(*
Nazwa:		FB_FormsDragStepper
Opis:		Przeciąganie formatek 
Wersja:		V0.22
Data:		2025-09-04
Autor:		DJ, DP
Urządzenia:	Siłownik podnoszenia wideł, Silnik krokowy przeciągania 
Ostatnie zmiany:
	- 20250904 [DP] EventLog->wywołać błędy 
	- 2025-08-19 [DP] Homing false
	- 2024-11-25 [DP] Czujnik dół
	- 2024-10-01 [DP] ESTOP Delay
	- RRRR-MM-DD [KTO?] Tekst Tekst Tekst Tekst Tekst Tekst Tekst Tekst Tekst Tekst 
	- 2025-09-15[VS] Jazda i stop w pozycji końcowej
Konfiguracja:
	- Krokówka
	Instukcja:
		-
		-
		-
	
Info:
	- Obsługa tylko jednego siłownika podnoszenia i dwóch siłowników prowadzących

*)

FUNCTION_BLOCK FB_FormsDragStepper
VAR_INPUT
	bEnable										: BOOL;				//Zezwolenie na pracę
	bEStop										: BOOL;				//Stop awaryjny włączony
	bRun										: BOOL;				//Rozkaz przeciagania
	bPrepare									: BOOL;				//Rozkaz przygotownaia 
	bDragUpWhenReady							: BOOL;					
	bHoming										: BOOL;				//Zezwolenie na wykonanie bazowania i pozycjonowanie układu
	bHomingDirection							: BOOL;				//Kierunek bazowania
	bBefore2ActuatorOff							: BOOL;
	bDelayAfterDrag								: BOOL;				//Opóżnienie po przeciąganiu
	bHeightSet									: BOOL;				//Ustaw do pozycji
	bIgnoreError								: BOOL;				//Ignorowanie błędów 
	bReset										: BOOL;				//Reset błędu, jeśli jest w stanie "eError"
	bResetCycle									: BOOL;				//Reset cyklu

	bTwoPhaseMode								: BOOL;				//Załączone dozowanie dwufazowe
	lrMinPosition								: LREAL;			 	
	lrMaxPosition								: LREAL;			 		
	lrStartPosition								: LREAL;			//Zadane położenie 
	lrMiddlePosition							: LREAL;			//Zadane położenie 
	lrEndPosition								: LREAL;			//Zadane położenie 		
	lrStartPositionTwoPhase						: LREAL;			//Zadane położenie 
	lrMiddlePositionTwoPhase					: LREAL;			//Zadane położenie 
	lrEndPositionTwoPhase						: LREAL;			//Zadane położenie 	
	lrLeadActuatorMoveUpPosition				: LREAL;			//Zadane położenie 	
	lrDragAcceleration							: LREAL;			//Przyspieszenie 
	lrDragDeceleration							: LREAL;			//Opóźnienie 
	lrDragJerk									: LREAL;			//Jerk
	lrDragSpeed									: LREAL;			//Prędkość 
	
	bHomingSensor								: BOOL;				//Czujnik bazowania 
	bDragUpSensor								: BOOL;				//
	bDragDownSensor								: BOOL;				//
	bLead1UpSensor								: BOOL;				//
	bLead2UpSensor								: BOOL;				//
	bManualMovement								: BOOL;				//Zezwolenie na ruchy ręczne

	_ALARMINFO_									: BOOL;
	iStationIndex								: UDINT;
	wsStationName								: WSTRING;
	bMoveToEndPosition							: BOOL;					//ustawienie w końcowej pozycji dla uruchomienia
END_VAR

VAR_OUTPUT
	eState										: E_Station;
	eRunningState								: E_DragStationState;	// Stan przeciągania formatek
	bError										: BOOL;					// Błąd stacji
	udiErrorID									: UDINT;				// Nr blędu przeciągania formatek
	sErrorDescription							: STRING(200);			// Opis błędu
	sErrorDescription2							: STRING(200);			// Opis błędu
	sErrorStationName							: STRING;				// Nazwa stacji
	udiStationID								: UDINT;				// Nr stacji

	bDragActuator								: BOOL;					
	bLeadBefore1Actuator						: BOOL;					
	bLeadBefore2Actuator						: BOOL;					
	
	bCycleDone									: BOOL;					//Sygnał zakończenia cyklu
	bCycleNotDone								: BOOL;
	bHomingDone									: BOOL;
	tCycleTime									: TIME;					//Czas cyklu
	lrActualDragPosition						: LREAL;				//Aktualne położenie
	//Dodatkowe	
	eRunningStateBeforeEStop					: E_DragStationState;	//Stan przed E-Stopem	
	bWasErrorOrEstop							: BOOL;
	
END_VAR

VAR
	(*LastStates*)
	eLastState									: E_Station;						//Stan ogólny bloku
	eLastStateTemp								: E_Station;						//Stan ogólny bloku
	eLastRunningState							: E_DragStationState;				//Stan podbloku
	eLastRunningStateTemp						: E_DragStationState;				//Stan podbloku
	
	(*Axis online*)
	fbDrag										: FB_McAxisOnlineNC;
	stDrag										: ST_McAxisOnline;
	                                    		                                 		
	(*Control*)
	tonResetting								: TON;								//Czas resetu
	tonHoming									: TON;
	tonPreparingToReady							: TON;								//Czas potrzeby na przygotowanie osi
	rtResetCommands								: R_TRIG;                                    	
	rtResetCycle								: R_TRIG;

	(*Statistics*)
	tonCycleTimer								: TON;								//Czas cyklu przeciągania	
	rtrigCycleTimerRead							: R_TRIG;

	(*Homing*)
	iHomingCase									: INT;
	
	(*Aborting*)
	iAbortingCase								: INT;
	                                    	
	(*Errors*)
	bStateError									: BOOL;
	tonEstopDelay								: TON;
	bResetCycleOn								: BOOL;
	tonbDragUpSensor							: TON;	
	tonbDragDownSensor							: TON;		
	tonbLead1UpSensor							: TON;
	tonbLead2UpSensor							: TON;
	
	(*Running*)

	tonNotDragActuatorDelay						: TON;
	tonRunningDraging							: TON;
	tonRunningeEndingOfDrag						: TON;
	(*Inne*)
	
		//Zmienne od EVENTLOGGER
	bAlarmInit 						: BOOL := TRUE; 
	nAlarmNumerator					: INT;
	arfbAlarm						: ARRAY[0..19] OF  FB_TcAlarm;		//Tablica bloczków błędów
	fbSourceInfo 					: FB_TcSourceInfo;
	iSourceInfo						: I_TcSourceInfo;
	sAlarmTest						: STRING;
	//Koniec zmiennych od EVENTLOGGER
	
END_VAR
	
VAR_IN_OUT
	bManualDragActuator							: BOOL;		
	bManualLeadBefore1Actuator					: BOOL;			
	bManualLeadBefore2Actuator					: BOOL;			
	bManualDragRight							: BOOL;				
	bManualDragLeft								: BOOL;		
	DragAxisRef									: AXIS_REF;		
END_VAR

ResetAll();
ErrorHandling();
Signals();
Control();
Limits();
DragControlBlocks();
Statistics();
aStationID();
(*Zapisywanie ostatniego stanu*)
IF eLastStateTemp<>eState THEN
	eLastState := eLastStateTemp;
END_IF
eLastStateTemp := eState;
IF eLastRunningStateTemp<>eRunningState THEN
	eLastRunningState := eLastRunningStateTemp;
END_IF
eLastRunningStateTemp := eRunningState;
(*Koniec Zapisywanie ostatniego stanu*)

ACTION aStationID:
udiStationID	:=	iStationIndex;
END_ACTION

ACTION Control:


	(*****Wyłączenie enable*****)
	IF NOT bEnable AND NOT bError THEN
		IF eState <> E_Station.eDisabled AND eState <> E_Station.ePreparingToDisable THEN
				eState 								:= E_Station.ePreparingToDisable; 
		END_IF	
	END_IF

	(*****Estop*****)
	IF NOT bEstop  THEN	
		IF eState <> E_Station.eAborted AND eState <> E_Station.eAborting AND eState <> E_Station.eDisabled THEN
				eRunningStateBeforeEStop			:= eRunningState;
				eState 								:= E_Station.eAborting; 
				iAbortingCase						:= 0; 
		END_IF
	END_IF


	
CASE eState OF
	
//==========================================================================================	
	E_Station.eDisabled: 						// Stan nieaktywnosci (Stacja wyłączona) 
		
		IF bEnable THEN
			eState 									:= E_Station.ePreparingToReady; 
		END_IF 

//==========================================================================================	    
	E_Station.eAborted: 						// Stan bezpiecznego zatrzymania (po Abortingu) 	
			
		IF bEStop THEN
			bWasErrorOrEstop						:= TRUE;	
			eState 									:= E_Station.ePreparingToReady;
		END_IF		
			
//==========================================================================================	
	E_Station.eAborting:                 		// Stan bezpiecznego zatrzymywania (po EStopie)
		
		CASE iAbortingCase OF
			
			0: //Inicjalizacja
				IF stDrag.mcPower.bStatus THEN
					iAbortingCase					:= 10;
				ELSE
					iAbortingCase					:= 40;
				END_IF
				
			10: //Komenda MC_STOP
				stDrag.mcStop.bExecute				:= TRUE;	
				//Czekam na Done
				IF stDrag.mcStop.bDone THEN
					stDrag.mcStop.bExecute			:= FALSE;
					iAbortingCase					:= 20;
				END_IF
				
			20: //Kasowanie komend
				stDrag.mcMoveAbsolute.bExecute		:= FALSE;
				stDrag.mcMoveRelative.bExecute		:= FALSE;
				ResetCommands();
				iAbortingCase						:= 30;
	
			30: //Wyłączenie osi
				stDrag.mcPower.bEnable				:= FALSE;
				stDrag.mcPower.bEnable_Negative		:= FALSE;
				stDrag.mcPower.bEnable_Positive		:= FALSE;
				IF NOT stDrag.mcPower.bStatus THEN
					iAbortingCase					:= 40;
				END_IF
				
			40: //Kasowanie podzespołow
				ResetCommands();
				iAbortingCase						:= 50;
				
			50: //Przejście do Aborted
				iAbortingCase						:= 0;
				eState								:= E_Station.eAborted;
				eRunningState						:= E_DragStationState.eReady;
				
		END_CASE

//==========================================================================================			
	E_Station.eError:                 	 		// Stan błędu 	
		
		bWasErrorOrEstop							:= TRUE;

		IF bReset THEN
			eState									:= E_Station.eResetting;	
		ELSE
			ResetCommands();
		END_IF
			
//==========================================================================================
	E_Station.eResetting:						// Stan resetowania bledu (po Errorze)
			
	//Procedura obsługi resetu w zależności od błędu
//	CASE udiErrorID OF 
//	CASE udiErrorID - iStationIndex(*udiResetStep*) OF 	
//		171: //Error 1 - Błąd Serwa
		IF  arfbAlarm[0].bActive THEN
			stDrag.mcReset.bExecute					:= TRUE;
			IF stDrag.mcReset.bDone THEN
				stDrag.mcReset.bExecute				:= FALSE;
				bError								:= FALSE;
			END_IF	
		END_IF
		
//		172,173://Error 2 - Błąd siłownika przeciągania
		IF  arfbAlarm[1].bActive OR arfbAlarm[2].bActive THEN
			bDragActuator							:= FALSE;	
			//bLeadBefore1Actuator					:= FALSE;				
			//bLeadBefore2Actuator					:= FALSE;			
			bError									:= FALSE;
		END_IF	
// 		174: //Error 4 - Błąd siłownika prowadzenia
		IF arfbAlarm[3].bActive THEN
			//bDragActuator							:= FALSE;	
			bLeadBefore1Actuator					:= TRUE;				
			//bLeadBefore2Actuator					:= FALSE;			
			bError									:= FALSE;		
		END_IF
// 		175: //Error 5 - Błąd siłownika prowadzenia
		IF arfbAlarm[4].bActive THEN
			//bDragActuator							:= FALSE;	
			bLeadBefore2Actuator					:= NOT bBefore2ActuatorOff;				
			//bLeadBefore2Actuator					:= FALSE;			
			bError									:= FALSE;		
		END_IF
//	END_CASE
	
	IF NOT bError THEN
		udiErrorID									:= 0;
		sErrorDescription							:= '';
		sErrorDescription2							:= '';	
		eState										:= E_Station.ePreparingToReady;
	ELSIF tonResetting.Q THEN                   	
		eState										:= E_Station.eError;
	END_IF	
 
//==========================================================================================
	E_Station.eManualMovement:     				// Stan ruchów manualnych  
       
		ManualMovements();
		//Wyjście z trybu serwisowego
		IF NOT bManualMovement THEN
			bDragActuator							:=	bManualDragActuator;	
			bLeadBefore1Actuator					:=	bManualLeadBefore1Actuator;
			bLeadBefore2Actuator					:=	bManualLeadBefore2Actuator;
			eState									:=	E_Station.eReady;
		END_IF 

//==========================================================================================		
	E_Station.eHoming:							// Stan bazowania 
		
		Homing();	
		IF NOT bHoming AND NOT bHeightSet AND tonHoming.Q THEN
			eState									:=	E_Station.ePreparingToReady;
		END_IF		
			
//==========================================================================================
	E_Station.eHomingDone:                  	// Stan wykonania bazowania 

		bHomingDone									:= TRUE;
		bResetCycleOn								:= FALSE;		
		IF NOT bHoming AND NOT bHeightSet AND NOT bResetCycleOn THEN
		//	eState									:=	E_Station.eReady;
			eState									:=	E_Station.ePreparingToReady;
		END_IF

//==========================================================================================
	E_Station.ePreparingToReady:            	// Stan przygotowywania do gotowosci (zawsze przed Ready)  

		IF tonPreparingToReady.Q THEN
			
			stDrag.mcPower.bEnable					:= TRUE;
			stDrag.mcPower.bEnable_Negative			:= TRUE;
			stDrag.mcPower.bEnable_Positive			:= TRUE;
			stDrag.mcPower.lrOverride				:= 100;
			
			IF stDrag.mcPower.bStatus THEN
				
				ResetCommands();
				eState								:= E_Station.eReady;
				eRunningState						:= E_DragStationState.eReady;
				
				IF bResetCycleOn THEN
					eState							:= E_Station.eHoming;
				END_IF
				
			END_IF
		
		END_IF			

//==========================================================================================
	E_Station.ePreparingToDisable:         	 	// Stan przygotowywania do nieaktywnosci (po wyłączeniu Enable) 
  
		stDrag.mcPower.bEnable						:= FALSE;
		stDrag.mcPower.bEnable_Negative				:= FALSE;
		stDrag.mcPower.bEnable_Positive				:= FALSE;
		stDrag.mcPower.lrOverride					:= 0;
		
		bWasErrorOrEstop							:= FALSE;
		bHomingDone									:= FALSE;	
		
		IF NOT stDrag.mcPower.bStatus THEN
			ResetCommands();
			eState									:= 	E_Station.eDisabled;
			eRunningState							:= 	E_DragStationState.eReady;
		END_IF

//==========================================================================================	
	E_Station.eReady:							// Stan gotowosci 


		(*Skasowanie wszystkich komend*)
		IF rtResetCommands.Q THEN	ResetCommands();	END_IF		
		
		IF bDragUpWhenReady THEN
			bDragActuator							:=	TRUE;
		END_IF
	
		IF (bRun OR bPrepare) AND NOT bCycleDone THEN
			eState									:= E_Station.eStarting;
			//IF bDragUpWhenReady THEN
				bDragActuator						:=	FALSE;
			//END_IF			
		END_IF		
		IF bHoming OR bHeightSet THEN
			eState									:= E_Station.eHoming;
		END_IF
		IF bManualMovement THEN
			bManualDragActuator						:=	bDragActuator;			
			bManualLeadBefore1Actuator				:=	bLeadBefore1Actuator;	
			bManualLeadBefore2Actuator				:=	bLeadBefore2Actuator;	
			bManualDragRight						:=	FALSE;		
			bManualDragLeft							:=	FALSE;					
			eState									:= E_Station.eManualMovement;					
		END_IF
		IF NOT bRun AND NOT bPrepare THEN
			bCycleDone								:= FALSE;
		END_IF

//==========================================================================================
	E_Station.eStopping:					// Stan zatrzymywania 
		
		Running();
		
		//Czekam dopóki skończy ruch
		IF	eRunningState <> E_DragStationState.eDraging AND eRunningState <> E_DragStationState.eDragingDone AND eRunningState <> E_DragStationState.eEndingOfDrag AND eRunningState <> E_DragStationState.eDraged
		AND  eRunningState <> E_DragStationState.eEndingOfDragDone AND  eRunningState <> E_DragStationState.eLowering  THEN	
			stDrag.mcReset.bExecute					:= TRUE;	
		END_IF
		
		//Reset ruchu
		IF stDrag.mcReset.bDone THEN		
			stDrag.mcReset.bExecute					:= FALSE;
			eState 									:= E_Station.eReady;
		END_IF

//==========================================================================================
	E_Station.eStarting:                  	// Stan uruchamiania (po Ready)
		
		eState										:= E_Station.eRunning;

//==========================================================================================
	E_Station.eRunning:               		// Stan wykonywania cyklu (po Startingu), w tym stanie osobny
 
		Running();

		IF NOT bRun AND NOT bPrepare THEN					(*Przerywanie cyklu*)
			eState 				 					:= E_Station.eStopping;	
		END_IF
			
		IF bCycleDone THEN (*Cykl zakończony*)
			eState 				 					:= E_Station.eReady;
		END_IF	
		
//==========================================================================================
END_CASE
END_ACTION

ACTION DragControlBlocks:
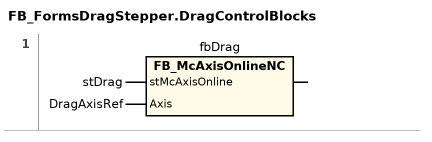
// NETWORK 1
fbDrag(stMcAxisOnline := stDrag, Axis := DragAxisRef); // FB_McAxisOnlineNC
END_ACTION

ACTION ErrorHandling:
// Alarm_0260	260	Error	Błąd napędu przeciągania. Błąd NC: {0}
// Alarm_0261	261	Error	Siłownik przeciągania | Blokada podnoszenia - sprawdź czujnik lub odblokuj
// Alarm_0262	262	Error	Siłownik przeciągania | Blokada opuszczania siłownika - sprawdź czujnik lub odblokuj
// Alarm_0263	263	Error	Siłownik prowadzenia | Blokada podnoszenia - sprawdź czujnik lub odblokuj
// Alarm_0264	264	Error	Siłownik prowadzenia | Blokada podnoszenia - sprawdź czujnik lub odblokuj

IF bAlarmInit THEN
    bAlarmInit := FALSE; 
	fbSourceInfo.Clear();
	fbSourceInfo.sName:=wsLiteral_TO_UTF8(wsStationName);//'Machine';
	fbSourceInfo.nId:=iStationIndex;//2700;
	// Alarm_0260	260	Error	Błąd napędu przeciągania. Błąd NC: {0}
    arfbAlarm[0].CreateEx(stEventEntry := TC_EVENTS.AlarmClass.Alarm_0260, bWithConfirmation:= FALSE,  ipSourceInfo:= fbSourceInfo); 
	// Alarm_0261	261	Error	Siłownik przeciągania | Blokada podnoszenia - sprawdź czujnik lub odblokuj
	arfbAlarm[1].CreateEx(stEventEntry := TC_EVENTS.AlarmClass.Alarm_0261, bWithConfirmation:= FALSE,  ipSourceInfo:= fbSourceInfo);
	// Alarm_0262	262	Error	Siłownik przeciągania | Blokada opuszczania siłownika - sprawdź czujnik lub odblokuj
	arfbAlarm[2].CreateEx(stEventEntry := TC_EVENTS.AlarmClass.Alarm_0262, bWithConfirmation:= FALSE,  ipSourceInfo:= fbSourceInfo);
	// Alarm_0263	263	Error	Siłownik prowadzenia | Blokada podnoszenia - sprawdź czujnik lub odblokuj
	arfbAlarm[3].CreateEx(stEventEntry := TC_EVENTS.AlarmClass.Alarm_0263, bWithConfirmation:= FALSE,  ipSourceInfo:= fbSourceInfo);
	// Alarm_0264	264	Error	Siłownik prowadzenia | Blokada podnoszenia - sprawdź czujnik lub odblokuj
	arfbAlarm[4].CreateEx(stEventEntry := TC_EVENTS.AlarmClass.Alarm_0264, bWithConfirmation:= FALSE,  ipSourceInfo:= fbSourceInfo);

	
END_IF

//CZYTANIE STATUSÓW
DragAxisRef.ReadStatus();

bStateError										:= (eState=E_Station.eError) OR (eState=E_Station.eResetting) OR NOT bEstop OR bIgnoreError;
tonEstopDelay									(IN:=bEStop,	PT:=T#4S);

IF bEnable AND tonEstopDelay.Q THEN
	// Alarm_0260	260	Error	Błąd napędu przeciągania. Błąd NC: {0}
	//Error 1 - Błąd Serwa
	IF stDrag.bError THEN
		bHomingDone									:= FALSE;	
		arfbAlarm[0].ipArguments.Clear() .AddString(stDrag.stError.sNcError);
		IF NOT arfbAlarm[0].bActive THEN
			stDrag.mcReset.bExecute				:= TRUE; // na testy jak wystąpi błąd
			arfbAlarm[0].Raise(nTimeStamp:=0);
		END_IF
	ELSE	
		IF  arfbAlarm[0].bActive AND bReset THEN
			arfbAlarm[0].Clear(nTimeStamp:=0, bResetConfirmation:= FALSE);
		END_IF	
// 		stDrag.mcReset.bExecute				:= TRUE; // na testy jak wystąpi błąd
// 		bError								:= TRUE;
// 		udiErrorID							:= 171;
// 		//udiErrorID							:= udiErrorID + iStationIndex;
// 		sErrorDescription					:= 'Błąd napędu przeciągania. Błąd NC:';
// 		sErrorDescription2					:= stDrag.stError.sNcError;
	END_IF
	
	//Alarm_0261	261	Error	Siłownik przeciągania | Blokada podnoszenia - sprawdź czujnik lub odblokuj
	//Error 2 - Błąd siłownika przeciągania
	tonbDragUpSensor	(IN:= bDragActuator AND NOT bDragUpSensor	, PT:=T#2S);
	IF tonbDragUpSensor.Q THEN
		bHomingDone									:= FALSE;			
		IF NOT arfbAlarm[1].bActive THEN
			arfbAlarm[1].Raise(nTimeStamp:=0);
		END_IF
	ELSE	
		IF  arfbAlarm[1].bActive AND bReset THEN
			arfbAlarm[1].Clear(nTimeStamp:=0, bResetConfirmation:= FALSE);
		END_IF	
// 		bError								:= TRUE;
// 		udiErrorID							:= 172;	
// 		//udiErrorID 							:= udiErrorID + iStationIndex;
// 		sErrorDescription					:= 'Siłownik przeciągania';
// 		sErrorDescription2					:= 'Blokada podnoszenia - sprawdź czujnik lub odblokuj';
	END_IF
	
	// Alarm_0262	262	Error	Siłownik przeciągania | Blokada opuszczania siłownika - sprawdź czujnik lub odblokuj
	//Error 3 - Błąd siłownika przeciągania
	tonbDragDownSensor	(IN:= NOT bDragActuator AND NOT bDragDownSensor	AND bRun, PT:=T#2S);
	IF tonbDragDownSensor.Q THEN
		IF NOT arfbAlarm[2].bActive THEN
			arfbAlarm[2].Raise(nTimeStamp:=0);
		END_IF
	ELSE	
		IF  arfbAlarm[2].bActive AND bReset THEN
			arfbAlarm[2].Clear(nTimeStamp:=0, bResetConfirmation:= FALSE);
		END_IF	
// 		bError								:= TRUE;
// 		udiErrorID							:= 173;	
// 		//udiErrorID 							:= udiErrorID + iStationIndex;
// 		sErrorDescription					:= 'Siłownik przeciągania';
// 		sErrorDescription2					:= 'Blokada opuszczania siłownika - sprawdź czujnik lub odblokuj';
	END_IF;			
	
	// Alarm_0263	263	Error	Siłownik prowadzenia | Blokada podnoszenia - sprawdź czujnik lub odblokuj
	//Error 4 - Błąd siłownika prowadzenia
	tonbLead1UpSensor	(IN:= bLeadBefore1Actuator AND NOT bLead1UpSensor	, PT:=T#2S);
	IF tonbLead1UpSensor.Q THEN
		IF NOT arfbAlarm[3].bActive THEN
			arfbAlarm[3].Raise(nTimeStamp:=0);
		END_IF
	ELSE	
		IF  arfbAlarm[3].bActive AND bReset THEN
			arfbAlarm[3].Clear(nTimeStamp:=0, bResetConfirmation:= FALSE);
		END_IF	
// 		bError								:= TRUE;
// 		udiErrorID							:= 174;	
// 		//udiErrorID 							:= udiErrorID + iStationIndex;
// 		sErrorDescription					:= 'Siłownik prowadzenia';
// 		sErrorDescription2					:= 'Blokada podnoszenia - sprawdź czujnik lub odblokuj';
	END_IF;		
	
	//// Alarm_0264	264	Error	Siłownik prowadzenia | Blokada podnoszenia - sprawdź czujnik lub odblokuj
	//Error 5 - Błąd siłownika prowadzenia
	tonbLead2UpSensor	(IN:= bLeadBefore2Actuator AND NOT bLead2UpSensor	, PT:=T#2S);
	IF tonbLead2UpSensor.Q THEN
		IF NOT arfbAlarm[4].bActive THEN
			arfbAlarm[4].Raise(nTimeStamp:=0);
		END_IF
	ELSE	
		IF  arfbAlarm[4].bActive AND bReset THEN
			arfbAlarm[4].Clear(nTimeStamp:=0, bResetConfirmation:= FALSE);
		END_IF	
// 		bError								:= TRUE;
// 		udiErrorID							:= 175;	
// 		//udiErrorID 							:= udiErrorID + iStationIndex;
// 		sErrorDescription					:= 'Siłownik prowadzenia';
// 		sErrorDescription2					:= 'Blokada podnoszenia - sprawdź czujnik lub odblokuj';
	END_IF;		
ELSE
	bError := FALSE;
END_IF

//******************PRZEJŚCIE DO eERROR*****************************

IF bError AND  NOT bStateError THEN
	eState 									:= E_Station.eError;
END_IF

//****************WYŚWIETLANIE STATUSU BLEDU************************
(*Wyświetlanie błedu na wyjściu*)
bError							:= FALSE;
FOR nAlarmNumerator := 0 TO 19 DO
	bError						:= bError OR arfbAlarm[nAlarmNumerator].bActive;
END_FOR

(*Przepisywanie nazwy stacji*)
sErrorStationName 							:= WSTRING_TO_STRING(wsStationName);
END_ACTION

ACTION Homing:

stDrag.mcMoveRelative.lrAcceleration			:=	1500;
stDrag.mcMoveRelative.lrDeceleration			:=	1500;
stDrag.mcMoveRelative.lrJerk					:=	15000;
stDrag.mcMoveRelative.lrVelocity				:=	15;

stDrag.mcMoveVelocity.lrAcceleration			:= 	2500;
stDrag.mcMoveVelocity.lrDeceleration			:= 	2500;
stDrag.mcMoveVelocity.lrJerk					:= 	2500;
stDrag.mcMoveVelocity.lrVelocity				:= 	10;	

stDrag.stStatus.lrPosDiff;
stdrag.stStatus.lrActPos;

IF bHoming THEN // Bazowanie - podjazd do góry i ustawienie obrotu
	CASE iHomingCase OF
	
	0: //Opuszczamy widły
		bHomingDone										:= FALSE;
		                                        		
		stDrag.mcMoveAbsolute.bExecute					:= FALSE;
		stDrag.mcMoveRelative.bExecute					:= FALSE;
		stDrag.mcMoveVelocity.bExecute					:= FALSE;
		
		bDragActuator									:= FALSE;	
		bLeadBefore1Actuator							:= TRUE; 	
		bLeadBefore2Actuator							:= NOT bBefore2ActuatorOff;
			
		iHomingCase										:= 10;
	
	10: //Sprawdzamy czy jest na czujniku
		IF bHomingSensor THEN
			iHomingCase									:= 20;
		ELSE                                        	
			iHomingCase									:= 30;
		END_IF
		
	20: //Muszę wyjechać z czujnika
		stDrag.mcMoveRelative.lrAcceleration			:=1500;
		stDrag.mcMoveRelative.lrDeceleration			:=1500;
		stDrag.mcMoveRelative.lrJerk					:=15000;
		stDrag.mcMoveRelative.lrVelocity				:=15;

		stDrag.mcMoveRelative.lrDistance				:= 50; // bylo 50
		IF bHomingDirection THEN
			stDrag.mcMoveRelative.lrDistance			:= -50; // bylo 50
		END_IF
		
		stDrag.mcMoveRelative.bExecute					:= TRUE;
		
		IF stDrag.mcMoveRelative.bDone THEN
			stDrag.mcMoveRelative.bExecute				:= FALSE;
			iHomingCase									:= 30;
		END_IF
		
	30: //Bazuje na czujnik
		stDrag.mcMoveVelocity.lrAcceleration			:= 2500;
		stDrag.mcMoveVelocity.lrDeceleration			:= 2500;
		stDrag.mcMoveVelocity.lrJerk					:= 2500;
		stDrag.mcMoveVelocity.lrVelocity				:= 10;	
	
		stDrag.mcMoveVelocity.eDirection				:= MC_Negative_Direction;
		IF bHomingDirection THEN
			stDrag.mcMoveVelocity.eDirection			:= MC_Positive_Direction;
		END_IF
		
		stDrag.mcMoveVelocity.bExecute					:= TRUE;
		
		IF bHomingSensor THEN
			stDrag.mcMoveVelocity.bExecute				:= FALSE;
			iHomingCase									:= 40;
		END_IF
		
	40: //Zatrzymanie osi
		stDrag.mcStop.bExecute							:= TRUE;
		
		IF stDrag.mcStop.bDone THEN
			stDrag.mcStop.bExecute						:= FALSE;
			iHomingCase									:= 50;
		END_IF
	
	50: 

		iHomingCase										:= 60;
		
	60: //Bazujemy Enkoder
		stDrag.mcHome.eHomingMode						:= MC_Direct;
		stDrag.mcHome.lrPosition						:= lrMinPosition;
		IF bHomingDirection THEN
			stDrag.mcHome.lrPosition					:= lrMaxPosition;
		END_IF
		
		stDrag.mcHome.bExecute							:= TRUE;
		                                        		
		IF stDrag.mcHome.bDone THEN             		
			stDrag.mcHome.bExecute						:= FALSE;
			iHomingCase									:= 70;
		END_IF
		
	70:                             	
		iHomingCase										:= 80;

	80:
		stDrag.mcMoveAbsolute.lrAcceleration			:=1500;
		stDrag.mcMoveAbsolute.lrDeceleration			:=1500;
		stDrag.mcMoveAbsolute.lrJerk					:=15000;
		stDrag.mcMoveAbsolute.lrVelocity				:=15;
									  
		stDrag.mcMoveAbsolute.lrPosition			  	:= lrStartPosition;
		stDrag.mcMoveAbsolute.bExecute				  	:= TRUE;
			
		IF stDrag.mcMoveAbsolute.bDone THEN
			stDrag.mcMoveAbsolute.bExecute				:= FALSE;
			iHomingCase									:= 100;
		END_IF	
		
	100: //Zbazowano	
		iHomingCase										:= 0;
		eState											:= E_Station.eHomingDone;
	
	END_CASE
END_IF	
IF bHeightSet THEN

	bDragActuator									:= FALSE;	
	bLeadBefore1Actuator							:= FALSE;	
	bLeadBefore2Actuator							:= FALSE;

	//Dynamika Ruchu
	stDrag.mcMoveAbsolute.lrAcceleration			:= lrDragAcceleration;
	stDrag.mcMoveAbsolute.lrDeceleration			:= lrDragDeceleration;
	stDrag.mcMoveAbsolute.lrVelocity				:= lrDragSpeed;
	stDrag.mcMoveAbsolute.lrJerk					:= 10000;
	                                            	                     	
	stDrag.mcMoveAbsolute.lrPosition				:= lrStartPosition;                                            	
	stDrag.mcMoveAbsolute.bExecute					:= TRUE;
	                                            	
	IF stDrag.mcMoveAbsolute.bDone THEN         	
		stDrag.mcMoveAbsolute.bExecute				:= FALSE;
		eState										:= E_Station.eHomingDone;
	END_IF
		
END_IF
END_ACTION

ACTION Limits:
(*Wywowyłanie na początku*)


(*Prędkość zakręcania*)


(*Inny parametr*)
//...
END_ACTION

ACTION ManualMovements:

IF NOT bRun AND NOT bPrepare AND bManualMovement THEN
	stDrag.mcJog.bJogForward						:=	bManualDragRight AND	lrActualDragPosition < lrEndPosition AND NOT bLeadBefore1Actuator;
	stDrag.mcJog.bJogBackwards						:=	bManualDragLeft AND		lrActualDragPosition > lrStartPosition AND NOT bLeadBefore1Actuator;                                  	                                  	                                   	
	bDragActuator									:=	bManualDragActuator;			
	bLeadBefore1Actuator							:=	bManualLeadBefore1Actuator;	
	bLeadBefore2Actuator							:=	bManualLeadBefore2Actuator;	
ELSE
	bManualDragActuator								:=	FALSE;		
	bManualLeadBefore1Actuator						:=	FALSE;		
	bManualLeadBefore2Actuator						:=	FALSE;		
END_IF
	
IF bHoming OR bHeightSet THEN
	eState											:=	E_Station.eHoming;	
END_IF                                                	

IF  (bRun OR bPrepare) AND bManualMovement THEN                                                     	
	Running();
END_IF

IF NOT bRun AND NOT bPrepare THEN
	bCycleDone 										:= FALSE;
	bCycleNotDone 									:= FALSE;	
END_IF
END_ACTION

ACTION ResetAll:
(*****Reset bloczka*****)
IF bEnable THEN
	IF eState <> E_Station.eDisabled AND eState <> E_Station.ePreparingToDisable THEN
		IF bResetCycle THEN
			bResetCycleOn						:= TRUE;
			eState								:= E_Station.ePreparingToReady;
		END_IF
	END_IF
END_IF


IF bResetCycleOn THEN
	
	ResetCommands();
	eRunningState							:= E_DragStationState.eReady;	
	eState 				 					:= E_Station.eReady;

END_IF
END_ACTION

ACTION ResetCommands:
//KAsowanie komend ruchu 
stDrag.mcJog.bJogForward								:=	FALSE;
stDrag.mcJog.bJogBackwards								:=	FALSE;
stDrag.mcHome.bExecute									:=	FALSE;
                                                          	
stDrag.mcMoveAbsolute.bExecute							:=	FALSE;
stDrag.mcMoveRelative.bExecute							:=	FALSE;
stDrag.mcMoveVelocity.bExecute							:=	FALSE;
                                                          	
stDrag.mcStop.bExecute									:=	FALSE;
stDrag.mcReset.bExecute									:=	FALSE;
                                                          	
bManualDragActuator										:=	FALSE;		
bManualLeadBefore1Actuator								:=	FALSE;	
bManualLeadBefore2Actuator								:=	FALSE;	
bManualDragRight										:=	FALSE;	
bManualDragLeft											:=	FALSE;	
                                                          	
bDragActuator											:=	FALSE;	
bLeadBefore1Actuator									:=	TRUE;	
bLeadBefore2Actuator									:=	NOT bBefore2ActuatorOff;
                                                          	
bResetCycleOn											:=	FALSE;	

iHomingCase												:=	0;
//bCycleDone								   				:=	FALSE;
END_ACTION

ACTION Running:
	
CASE eRunningState OF
	
	E_DragStationState.eDisabled:
		eRunningState								:= E_DragStationState.eReady; 
	
	E_DragStationState.eReady:
		IF NOT bMoveToEndPosition THEN
			IF NOT bCycleDone  THEN                                           	
				IF bRun OR bPrepare THEN   
					bDragActuator								:=	FALSE;
					eRunningState								:=	E_DragStationState.ePreparingToMove; 
       			END_IF
			END_IF
		ELSE
			bDragActuator								:=	TRUE;
			bLeadBefore1Actuator						:=	TRUE;
			bLeadBefore2Actuator						:=	TRUE;
			IF bRun OR bPrepare THEN   
					eRunningState								:=	E_DragStationState.ePreparingToMove; 
       			END_IF
		END_IF	
		//Po E-Stopie
(*		IF bWasErrorOrEstop THEN	
			bWasErrorOrEstop						:= FALSE;
			eRunningState							:= eRunningStateBeforeEStop;
		END_IF*)
		
// Sygnal przygotowania do przeciaganiecia formatek		
	E_DragStationState.ePreparingToMove:
	
		stDrag.mcMoveAbsolute.lrAcceleration		:= lrDragAcceleration;
		stDrag.mcMoveAbsolute.lrDeceleration		:= lrDragDeceleration;
		stDrag.mcMoveAbsolute.lrJerk				:= lrDragJerk;
		stDrag.mcMoveAbsolute.lrVelocity			:= lrDragSpeed;

		IF NOT bMoveToEndPosition THEN
			stDrag.mcMoveAbsolute.lrPosition			:= lrStartPosition;
			IF bTwoPhaseMode THEN //dwu-faza
				stDrag.mcMoveAbsolute.lrPosition		:= lrStartPositionTwoPhase;	
			END_IF	
	    	
			stDrag.mcMoveAbsolute.bExecute				:= TRUE;
        	
			IF stDrag.mcMoveAbsolute.bDone  THEN
				stDrag.mcMoveAbsolute.bExecute			:=	FALSE;
				eRunningState							:=	E_DragStationState.eLifting;
			END_IF                                      	                                              
		ELSIF bMoveToEndPosition AND NOT vis.bDosingTwoPhasesShow THEN
			stDrag.mcMoveAbsolute.lrPosition			:= lrEndPosition;
			stDrag.mcMoveAbsolute.bExecute				:= TRUE;
			eRunningState							:=	E_DragStationState.eLifting;
		ELSIF bMoveToEndPosition AND vis.bDosingTwoPhasesShow THEN
			stDrag.mcMoveAbsolute.lrPosition			:= lrEndPositionTwoPhase;
			stDrag.mcMoveAbsolute.bExecute				:= TRUE;
			eRunningState							:=	E_DragStationState.eLifting;	
		END_IF	
// Podnoszenie widel do przeciągania i sprawdzenie czy trafiły w otwór		
	E_DragStationState.eLifting:
	
		bDragActuator								:=	TRUE;		
		IF bDragUpSensor AND bRun THEN
			eRunningState							:=	E_DragStationState.eDraging;	
		END_IF
//  
	E_DragStationState.ePrepareToDrag:
		;
	
// Przeciąganie formatek
	E_DragStationState.eDraging:
	
		bLeadBefore1Actuator						:=	FALSE;	
		bLeadBefore2Actuator						:=	FALSE;
		
		IF NOT bTwoPhaseMode AND lrActualDragPosition > lrLeadActuatorMoveUpPosition THEN
			bLeadBefore1Actuator						:=	TRUE;	
		ELSIF bTwoPhaseMode AND lrActualDragPosition < (lrStartPositionTwoPhase - lrLeadActuatorMoveUpPosition) THEN
			bLeadBefore2Actuator						:=	TRUE;
		END_IF
			IF tonRunningDraging.Q THEN //100MS
				//Dynamika Ruchu
				stDrag.mcMoveAbsolute.lrAcceleration		:= lrDragAcceleration;
				stDrag.mcMoveAbsolute.lrDeceleration		:= lrDragDeceleration;
				stDrag.mcMoveAbsolute.lrJerk				:= lrDragJerk;
				stDrag.mcMoveAbsolute.lrVelocity			:= lrDragSpeed;
				
				IF NOT bMoveToEndPosition THEN
					stDrag.mcMoveAbsolute.lrPosition			:= lrMiddlePosition;
					IF bTwoPhaseMode THEN //dwu-faza
						stDrag.mcMoveAbsolute.lrPosition		:= lrMiddlePositionTwoPhase;	
					END_IF	
					stDrag.mcMoveAbsolute.bExecute				:= TRUE;
					IF stDrag.mcMoveAbsolute.bDone THEN
						stDrag.mcMoveAbsolute.bExecute			:= FALSE;
						eRunningState							:= E_DragStationState.eDragingDone;
					END_IF
				END_IF
	    IF bMoveToEndPosition AND NOT vis.bDosingTwoPhasesShow	THEN
			stDrag.mcMoveAbsolute.lrPosition			:= lrEndPosition;
			stDrag.mcMoveAbsolute.bExecute				:= TRUE;	
			IF stDrag.mcMoveAbsolute.bDone THEN
				stDrag.mcMoveAbsolute.bExecute			:= FALSE;
				bCycleDone								:= TRUE;
				eRunningState							:= E_DragStationState.eReady;
			END_IF
		ELSIF bMoveToEndPosition AND vis.bDosingTwoPhasesShow	THEN
			stDrag.mcMoveAbsolute.lrPosition			:= lrEndPositionTwoPhase;			
            stDrag.mcMoveAbsolute.bExecute				:= TRUE;	
            IF stDrag.mcMoveAbsolute.bDone THEN
            	stDrag.mcMoveAbsolute.bExecute			:= FALSE;
            	bCycleDone								:= TRUE;
            	eRunningState							:= E_DragStationState.eReady;
	        END_IF
		END_IF
		END_IF
		//Szybsze otwieranie prowadzeń ZA o 2mm szybciej ZA szlaban chaczy
		IF NOT bTwoPhaseMode AND lrActualDragPosition > (lrMiddlePosition - 2) THEN
			bLeadBefore2Actuator						:=	NOT bBefore2ActuatorOff;	
		ELSIF bTwoPhaseMode AND lrActualDragPosition < (lrMiddlePositionTwoPhase + 2) THEN
			bLeadBefore1Actuator						:=	TRUE;
		END_IF				
		
	E_DragStationState.eDragingDone:

		bLeadBefore1Actuator						:=	TRUE;
		bLeadBefore2Actuator						:=	NOT bBefore2ActuatorOff;		
		eRunningState								:= E_DragStationState.eEndingOfDrag;
	
	E_DragStationState.eEndingOfDrag:
	
		//Dynamika Ruchu
		stDrag.mcMoveAbsolute.lrAcceleration		:= lrDragAcceleration;
		stDrag.mcMoveAbsolute.lrDeceleration		:= lrDragDeceleration;
		stDrag.mcMoveAbsolute.lrJerk				:= lrDragJerk;		
		stDrag.mcMoveAbsolute.lrVelocity			:= lrDragSpeed;
		
		stDrag.mcMoveAbsolute.lrPosition			:= lrEndPosition;
		IF bTwoPhaseMode THEN //dwu-faza			//	3 +	(143 - 137) = 3 + 6 = 9
			stDrag.mcMoveAbsolute.lrPosition		:= lrEndPositionTwoPhase;	
		END_IF	
		stDrag.mcMoveAbsolute.bExecute				:= TRUE;
		
		IF stDrag.mcMoveAbsolute.bDone THEN
			
		 IF tonRunningeEndingOfDrag.Q OR NOT bDelayAfterDrag THEN //Opóżnienie na końcu ruchu z wysunietymi widłami
			stDrag.mcMoveAbsolute.bExecute			:= FALSE;
			eRunningState							:= E_DragStationState.eEndingOfDragDone;
		END_IF	
			
		END_IF
		
	E_DragStationState.eEndingOfDragDone:
		
		eRunningState								:= E_DragStationState.eLowering;
	
	E_DragStationState.eLowering:
	
		bDragActuator								:=	FALSE;		
		IF bDragDownSensor (*tonNotDragActuatorDelay.Q*) THEN
			eRunningState							:= E_DragStationState.eDraged;
		END_IF		

		
	E_DragStationState.eDraged:
	
		stDrag.mcMoveAbsolute.lrAcceleration		:= lrDragAcceleration;
		stDrag.mcMoveAbsolute.lrDeceleration		:= lrDragDeceleration;
		stDrag.mcMoveAbsolute.lrJerk				:= lrDragJerk;		
		stDrag.mcMoveAbsolute.lrVelocity			:= lrDragSpeed;
		
		stDrag.mcMoveAbsolute.lrPosition			:= lrStartPosition;
		IF bTwoPhaseMode THEN //dwu-faza			
			stDrag.mcMoveAbsolute.lrPosition		:= lrStartPositionTwoPhase;
		END_IF			
		
		stDrag.mcMoveAbsolute.bExecute				:= TRUE;
	
		IF stDrag.mcMoveAbsolute.bDone THEN
			stDrag.mcMoveAbsolute.bExecute			:= FALSE;
			eRunningState							:= E_DragStationState.eDragedDone;
		END_IF
		
	E_DragStationState.eDragedDone:
	
		bCycleDone									:= TRUE;	
		eRunningState								:= E_DragStationState.eReady;	
		
END_CASE
END_ACTION

ACTION Signals:

tonPreparingToReady		(IN:=	eState = E_Station.ePreparingToReady			,PT:= T#3S);
tonResetting			(IN:=	eState = E_Station.eResetting					,PT:= T#200MS);
tonHoming				(IN:=	eState = E_Station.eHoming						,PT:= T#1S);
rtResetCommands			(CLK:=	eState = E_Station.eReady 						,Q=>); 

tonRunningDraging		(IN:=	eRunningState = E_DragStationState.eDraging		,PT:= T#100MS);	//bylo 100
tonRunningeEndingOfDrag	(IN:=	eRunningState = E_DragStationState.eEndingOfDrag AND
								stDrag.mcMoveAbsolute.bDone
								,PT:= T#5MS);								//100ms t#200ms

//Opóżnienie wysuwania przeciągania
tonNotDragActuatorDelay	(IN:=	NOT bDragActuator					,PT:=T#150MS);

	
//Aktualna pozycja przeciągania
lrActualDragPosition:= stDrag.stStatus.lrActPos;


//
END_ACTION

ACTION Statistics:
rtrigCycleTimerRead(CLK:=bCycleDone);
IF rtrigCycleTimerRead.Q THEN
	tCycleTime:=tonCycleTimer.ET;
END_IF
tonCycleTimer(IN:= eRunningState>E_DragStationState.eReady, PT:=T#1D);
END_ACTION

END_FUNCTION_BLOCK

(* stored: Version 1.1.0.1, ProductVersion 3.1.4026.13, FileIdentifier 842e6930b5d49100b0c27ef1683a7c5c5e6a8125, FileSignature 694c922db6e2ad4ab9d475c1b1400df63b80b50c44d86bdad5bbe205693e4d243a5f79439f43cd822c53e547a08474f5fc4f19f7265ccfbb1950772397d92261850c497555ab6b8fafa0e7a37d67661c2cab36714ae71e66acf8142b32c83a13c3ac8b22d05b259d06910ee01c976fccf5d983b33c2a7b276a74c1da3176c615b7b4f91646e00e72968cd8669bd99c3438a3c4f4286c12546b2a3990b03a847246f418cd2a555632e54b48584c4f354756e319b23c95047ce5e1ab100fedd04d1d6d066a11033ef81f577b186dbaef498a8773f9f91bafc4a8b2a24c0a548621a04ef08de9039ab4ac57ca9d7d13359bd4b960e81c2659e18a20b3df5af31aa5
   POU FB_FormsDragStepper: Id {bd208d61-6781-4acf-8f11-6d387e0a13ff}, SpecialFunc None
   Action aStationID: Id {9ccd54f6-98d1-4938-b4d7-6b5d5ae1ca8a}
   Action Control: Id {cbc9d799-0c48-40b5-b7eb-9253263c1b81}
   Action DragControlBlocks: Id {b4bde060-d82c-4be7-adca-88f8c3e744af}
   Action ErrorHandling: Id {1366f01f-87ff-4d9b-bc8d-76db944f0898}
   Action Homing: Id {770e5245-bb7b-46f8-a1e2-193bcfad055b}
   Action Limits: Id {f01c0429-ae4b-4c6b-b2af-7fd92c549760}
   Action ManualMovements: Id {7e2670d7-ce86-43a3-9662-d82e8ef5dc0f}
   Action ResetAll: Id {9adf339d-3a32-46b0-aa31-f5d0742526f4}
   Action ResetCommands: Id {c5a32987-e16b-4466-9c37-dd8311479005}
   Action Running: Id {60c30774-153f-4947-9d00-d8f0a71268e9}
   Action Signals: Id {aec3cd52-c285-47b5-be0d-1eebe10ed94e}
   Action Statistics: Id {d6a01f07-b649-4758-bbc1-44ca8bdd597b} *)
